FUNCTION ADC_5V : REAL
VAR_INPUT
	normal_input : REAL;
	x_max : REAL := 4.5;
	x_min : REAL := 0.5;
END_VAR
VAR
	voltage_reading : REAL;
END_VAR

// 0.5 - 4.5V AI INPUT  | normal_input 0 - 100%
voltage_reading := 4.5 * normal_input;
ADC_5V := (voltage_reading - x_min) / (x_max - x_min);

END_FUNCTION

(* stored: Version 1.1.0.1, ProductVersion 3.1.4024.11
   POU ADC_5V: Id {3d67c97b-d51a-4a8a-a967-1811c00ef817}, SpecialFunc None *)
